// TIA Portal V19 export
ORGANIZATION_BLOCK "PID P-502"   // OB30, LAD, CyclicInterrupt
{ S7_Optimized_Access := 'TRUE' }
// stored: SetENOAutomatically false
   VAR_INPUT
      Initial_Call : Bool;   // Initial call of this OB
      Event_Count : Int;   // Events discarded
   END_VAR
BEGIN

REGION Network 1: enable mode
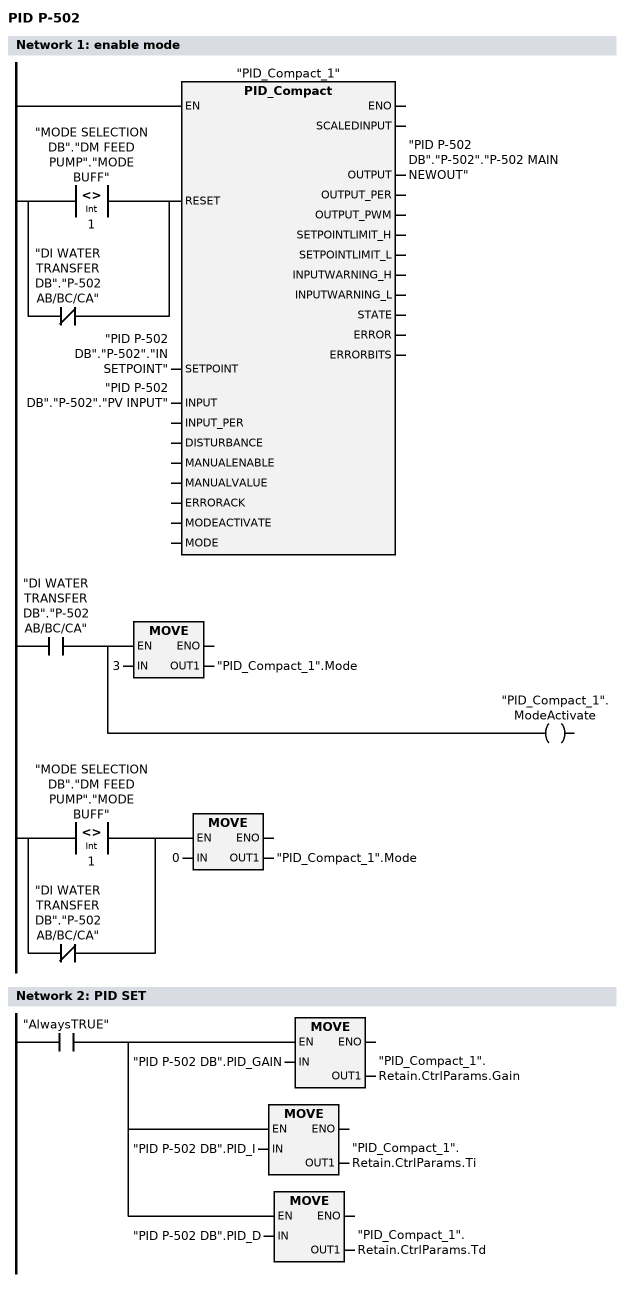
   RUNG wire#powerrail
      "PID_Compact_1".PID_Compact(Reset := wire#w1, Setpoint := "PID P-502 DB"."P-502"."IN SETPOINT", Input := "PID P-502 DB"."P-502"."PV INPUT", Input_PER :=, Disturbance :=, ManualEnable :=, ManualValue :=, ErrorAck :=, ModeActivate :=, Mode :=, ScaledInput =>, Output => "PID P-502 DB"."P-502"."P-502 MAIN NEWOUT", Output_PER =>, Output_PWM =>, SetpointLimit_H =>, SetpointLimit_L =>, InputWarning_H =>, InputWarning_L =>, State =>, Error =>, ErrorBits =>)
   END_RUNG
   RUNG wire#powerrail
      { S7_Templates := "SrcType := Int" } NE_Contact(in1 := "MODE SELECTION DB"."DM FEED PUMP"."MODE BUFF", in2 := 1)
   END_RUNG wire#w1
   RUNG wire#powerrail
      I_Contact( "DI WATER TRANSFER DB"."P-502 AB/BC/CA" )
   END_RUNG wire#w1
   RUNG wire#powerrail
      Contact( "DI WATER TRANSFER DB"."P-502 AB/BC/CA" )
      wire#w2
      Move(in := 3, out1 => "PID_Compact_1".Mode)
   END_RUNG
   RUNG wire#w2
      Coil( "PID_Compact_1".ModeActivate )
   END_RUNG
   RUNG wire#powerrail
      { S7_Templates := "SrcType := Int" } NE_Contact(in1 := "MODE SELECTION DB"."DM FEED PUMP"."MODE BUFF", in2 := 1)
      wire#w3
      Move(in := 0, out1 => "PID_Compact_1".Mode)
   END_RUNG
   RUNG wire#powerrail
      I_Contact( "DI WATER TRANSFER DB"."P-502 AB/BC/CA" )
   END_RUNG wire#w3
   // the same network as SCL:
   "PID_Compact_1"(Reset := ("MODE SELECTION DB"."DM FEED PUMP"."MODE BUFF" <> 1) OR NOT "DI WATER TRANSFER DB"."P-502 AB/BC/CA",   // PID_Compact
                   Setpoint := "PID P-502 DB"."P-502"."IN SETPOINT",
                   Input := "PID P-502 DB"."P-502"."PV INPUT",
                   Output => "PID P-502 DB"."P-502"."P-502 MAIN NEWOUT");
   IF "DI WATER TRANSFER DB"."P-502 AB/BC/CA" THEN "PID_Compact_1".Mode := 3; END_IF;
   "PID_Compact_1".ModeActivate := "DI WATER TRANSFER DB"."P-502 AB/BC/CA";
   IF ("MODE SELECTION DB"."DM FEED PUMP"."MODE BUFF" <> 1) OR NOT "DI WATER TRANSFER DB"."P-502 AB/BC/CA" THEN
       "PID_Compact_1".Mode := 0;
   END_IF;
END_REGION

REGION Network 2: PID SET
   RUNG wire#powerrail
      Contact( "AlwaysTRUE" )
      wire#w1
      Move(in := "PID P-502 DB".PID_GAIN, out1 => "PID_Compact_1".Retain.CtrlParams.Gain)
   END_RUNG
   RUNG wire#w1
      Move(in := "PID P-502 DB".PID_I, out1 => "PID_Compact_1".Retain.CtrlParams.Ti)
   END_RUNG
   RUNG wire#w1
      Move(in := "PID P-502 DB".PID_D, out1 => "PID_Compact_1".Retain.CtrlParams.Td)
   END_RUNG
   // the same network as SCL:
   IF "AlwaysTRUE" THEN
       "PID_Compact_1".Retain.CtrlParams.Gain := "PID P-502 DB".PID_GAIN;
       "PID_Compact_1".Retain.CtrlParams.Ti := "PID P-502 DB".PID_I;
       "PID_Compact_1".Retain.CtrlParams.Td := "PID P-502 DB".PID_D;
   END_IF;
END_REGION
END_ORGANIZATION_BLOCK
